PROGRAM AnalogConversion
VAR
	i					: INT := 1; //charger 1-8
	j					: INT := 1;  // section 1 - 4 
	k					: INT := 1;  // cap 1-10
	m					: INT := 1; //form cap 1-12
END_VAR

//Converting raw data into Voltage Reading (0-10V), (0.5-4.5V)   
//unfinish

//MCP Charger 
//Analog Input
//FOR i := 1 TO 8 BY 1 DO
FOR i := 1 TO 3 BY 1 DO
	
	MCP_IO.Charger[i].ChargerType_12kV := NOT MCP_IO.Charger[i].ChargerType_50kV;
	//voltage
	MCP_IO.Charger[i].voltageFeedback_norm := Norm_x (raw_input := INT_TO_REAL (MCP_IO.Charger[i].voltageFeedback_raw),
														x_max := 32767,
														x_min := 0);
	//current																									
	MCP_IO.Charger[i].currentFeedback_norm := Norm_x (raw_input := INT_TO_REAL (MCP_IO.Charger[i].currentFeedback_raw),
														x_max := 32767,
														x_min := 0);
	//50kV chargers feedback
	//if 50kV config selected
	IF MCP_IO.Charger[i].ChargerType_50kV = TRUE THEN 
		//50kv
		MCP_IO.Charger[i].voltageFeedback := (EngVal.Max_50kVChargerVoltage - EngVal.Min_50kVChargerVoltage) * ADC_10V(
																							normal_input := MCP_IO.Charger[i].voltageFeedback_norm,
																							x_max := 10,
																							x_min := 0);

		MCP_IO.Charger[i].currentFeedback := (EngVal.Max_50kVChargerCurrent - EngVal.Min_50kVChargerCurrent) * ADC_10V(
																							normal_input := MCP_IO.Charger[i].currentFeedback_norm,
																							x_max := 10,
																							x_min := 0);
		//12kv
	ELSIF MCP_IO.Charger[i].ChargerType_12kV = TRUE THEN
		MCP_IO.Charger[i].voltageFeedback := (EngVal.Max_12kVChargerVoltage - EngVal.Min_12kVChargerVoltage) * ADC_10V(
																							normal_input := MCP_IO.Charger[i].voltageFeedback_norm,
																							x_max := 10,
																							x_min := 0);
		MCP_IO.Charger[i].currentFeedback := (EngVal.Max_12kVChargerCurrent - EngVal.Min_12kVChargerCurrent) * ADC_10V(
																							normal_input := MCP_IO.Charger[i].currentFeedback_norm,
																							x_max := 10,
																							x_min := 0);										
	END_IF;	
END_FOR;

//Analog Output
//voltageSP = Required Charge Voltage******************
//limit for charing the cap
//FOR i := 1 TO 8 BY 1 DO
FOR i := 1 TO 3 BY 1 DO	
	//if 50kV config selected
	IF MCP_IO.Charger[i].ChargerType_50kV = TRUE THEN 
		//set limits of charger voltage input 
		IF MCP_IO.Charger[i].voltageSP >= REAL_TO_DINT (EngVal.UpperLimit50kVCaps) THEN
			MCP_IO.Charger[i].voltageSP := 35000; //limit at 35kV
		ELSIF MCP_IO.Charger[i].voltageSP <= 0 THEN
			MCP_IO.Charger[i].voltageSP := 0; //limit at 0V
		END_IF; 
		
	//prepare output signal for 50kV chargers.
		MCP_IO.Charger[i].voltageSP_norm := Norm_x (raw_input := DINT_TO_REAL (MCP_IO.Charger[i].voltageSP), 
												x_max := EngVal.Max_50kVChargerVoltage,
												x_min := EngVal.Min_50kVChargerVoltage);	
												
		MCP_IO.Charger[i].voltageSP_raw := AQ (norm_input := MCP_IO.Charger[i].voltageSP_norm, 
												x_max := 10,
												x_min := 0);
	END_IF;
		
	//if 12kV config selected
	IF MCP_IO.Charger[i].ChargerType_12kV = TRUE THEN
		//set limits of charger voltage input 
		IF MCP_IO.Charger[i].voltageSP <= 0 THEN
			MCP_IO.Charger[i].voltageSP := ABS(MCP_IO.Charger[i].voltageSP);
		END_IF
		
		IF MCP_IO.Charger[i].voltageSP >= REAL_TO_DINT (EngVal.UpperLimit12kVCaps) THEN
			MCP_IO.Charger[i].voltageSP := 10000; //limit at 10kV
		END_IF;

		//prepare output signal for 12kV chargers.
		MCP_IO.Charger[i].voltageSP_norm := Norm_x (raw_input := DINT_TO_REAL (MCP_IO.Charger[i].voltageSP), 
												x_max := EngVal.Max_12kVChargerVoltage,
												x_min := EngVal.Min_12kVChargerVoltage);
		
		MCP_IO.Charger[i].voltageSP_raw := AQ (norm_input := MCP_IO.Charger[i].voltageSP_norm, 
												x_max := 10,
												x_min := 0); 
	END_IF;	
												
	//limite for output sigal (<= 10V)  this should not happen
	IF MCP_IO.Charger[i].voltageSP_raw >= 32767 THEN 
		MCP_IO.Charger[i].voltageSP_raw := 32767; 										
	END_IF;
	
END_FOR;

//limits for gls 
IF MCP_IO.GLS1_voltageSP >= REAL_TO_DINT (EngVal.Max_GLS1_ChargerV) THEN 
	MCP_IO.GLS1_voltageSP := REAL_TO_DINT (EngVal.Max_GLS1_ChargerV);
	ELSIF MCP_IO.GLS1_voltageSP <= 0 THEN
		MCP_IO.GLS1_voltageSP := 0;
END_IF
IF MCP_IO.GLS2_voltageSP >= REAL_TO_DINT (EngVal.Max_GLS2_ChargerV) THEN 
	MCP_IO.GLS2_voltageSP := REAL_TO_DINT (EngVal.Max_GLS2_ChargerV);
	ELSIF MCP_IO.GLS2_voltageSP <= 0 THEN
		MCP_IO.GLS2_voltageSP := 0 ; 
END_IF
IF MCP_IO.GLS3_voltageSP >= REAL_TO_DINT (EngVal.ULimit_PreFormCapRequiredV) THEN 
	MCP_IO.GLS3_voltageSP := REAL_TO_DINT (EngVal.ULimit_PreFormCapRequiredV);
	ELSIF MCP_IO.GLS3_voltageSP <= 0 THEN
		MCP_IO.GLS3_voltageSP := 0 ; 
END_IF

//prepare analog output for gls chargers.	
MCP_IO.GLS1_voltageSP_norm := Norm_x (raw_input := DINT_TO_REAL (MCP_IO.GLS1_voltageSP),
									x_max := EngVal.Max_GLS1_ChargerV,
									x_min := 0);
MCP_IO.GLS1_voltageSP_raw:= AQ (norm_input := MCP_IO.GLS1_voltageSP_norm,
									x_max := 10,
									x_min := 0);									
									
MCP_IO.GLS2_voltageSP_norm := Norm_x (raw_input := DINT_TO_REAL (MCP_IO.GLS2_voltageSP),
									x_max := EngVal.Max_GLS2_ChargerV,
									x_min := 0);
MCP_IO.GLS2_voltageSP_raw:= AQ (norm_input := MCP_IO.GLS2_voltageSP_norm,
									x_max := 10,
									x_min := 0);	
									
MCP_IO.GLS3_voltageSP_norm := Norm_x (raw_input := DINT_TO_REAL (MCP_IO.GLS3_voltageSP),
									x_max := EngVal.Max_GLS3_ChargerV,
									x_min := 0);
MCP_IO.GLS3_voltageSP_raw:= AQ (norm_input := MCP_IO.GLS3_voltageSP_norm,
									x_max := 10,
									x_min := 0);	

//LCP 1 - 3 AI
FOR j := 1 TO 3 BY 1 DO 
	FOR k := 1 TO 10 BY 1 DO 
		LCP.Section[j].Peak.Cap[k].voltageFeedback_Norm := Norm_x (raw_input := INT_TO_REAL (LCP.Section[j].Peak.Cap[k].voltageFeedback_raw),
																x_max := 32767,
																x_min := 0);
																
		LCP.Section[j].Peak.Cap[k].voltageFeedback := (EngVal.Max_CapVoltage - EngVal.Min_CapVoltage) * ADC_10V (
																								normal_input := LCP.Section[j].Peak.Cap[k].voltageFeedback_Norm,
																								x_max := 10,
																								x_min := 0);
		//sustain caps 1 - 2
		LCP.Section[j].Sust.Cap[1].voltageFeedback_Norm := Norm_x (raw_input := INT_TO_REAL (LCP.Section[j].Sust.Cap[1].voltageFeedback_raw),
																x_max := 32767,
																x_min := 0);
																
		LCP.Section[j].Sust.Cap[1].voltageFeedback := (EngVal.Max_CapVoltage - EngVal.Min_CapVoltage) * ADC_10V (
																								normal_input := LCP.Section[j].Sust.Cap[1].voltageFeedback_Norm,
																								x_max := 10,
																								x_min := 0);
																
		LCP.Section[j].Sust.Cap[2].voltageFeedback_Norm := Norm_x (raw_input := INT_TO_REAL (LCP.Section[j].Sust.Cap[2].voltageFeedback_raw),
																x_max := 32767,
																x_min := 0);
																
		LCP.Section[j].Sust.Cap[2].voltageFeedback := (EngVal.Max_CapVoltage - EngVal.Min_CapVoltage) * ADC_10V (
																								normal_input := LCP.Section[j].Sust.Cap[2].voltageFeedback_Norm,
																								x_max := 10,
																								x_min := 0);
	END_FOR;	
END_FOR

//LCP 4 AI
FOR m := 1 TO 12 BY 1 DO
	LCP.Section[4].Form.Cap[m].voltageFeedback_norm := Norm_x (raw_input := INT_TO_REAL (LCP.Section[4].Form.Cap[m].voltageFeedback_raw),
																x_max := 32767,
																x_min := 0);
																
	LCP.Section[4].Form.Cap[m].voltageFeedback := (EngVal.Max_CapVoltage - EngVal.Min_CapVoltage) * ADC_10V (
																							normal_input := LCP.Section[4].Form.Cap[m].voltageFeedback_norm,
																							x_max := 10,
																							x_min := 0);
END_FOR;

//preform  cap AI
LCP.Section[4].PreFormCapVoltage_norm := Norm_x (raw_input := INT_TO_REAL (LCP.Section[4].PreFormCapVoltage_raw),
														x_max := 32767,
														x_min := 0);
															
LCP.Section[4].PreFormCapVoltageFeedback := (EngVal.Max_CapVoltage - EngVal.Min_CapVoltage) * ADC_10V (
																							normal_input := LCP.Section[4].PreFormCapVoltage_norm,
																							x_max := 10,
																							x_min := 0);															


//reset counter
//IF i > 8 THEN
IF i > 3 THEN
	i:=1;
END_IF;

IF j > 3 THEN 
	j := 1;
END_IF

IF k > 10 THEN 
	k := 1;
END_IF

IF m > 12 THEN 
	m := 1;
END_IF

END_PROGRAM

(* stored: Version 1.1.0.1, ProductVersion 3.1.4024.11
   POU AnalogConversion: Id {3b8eecca-a8e5-4cfd-bb8d-8865397a6f0b}, SpecialFunc None *)
